// TIA Portal V21 export
TYPE "OBJ_Washing_Phase_V100_Type"
   STRUCT
      x_Start_Ok : Bool;   // 0.2 - Consenso Inizio Fase
      x_EN_Next_Step : Bool;   // 0.3 - Abilita Passo Successivo (al pastorizzatore)
      Free04 : Bool;
      x_Aux_Next_Step_After_Drain : Bool;   // 0.5 - Aux Passo Successivo Dopo Drenaggio
      x_Start_Step_Mngr : Bool;   // 0.6 - InizioGestionePassi
      x_Stop_Step_Mngr : Bool;   // 0.7 - FineGestionePassi
      x_AppFP_Start : Bool;   // 1.0 - AppoggioFrInizio
      x_Pulse_Start : Bool;   // 1.1 - FronteInizio
   END_STRUCT;
END_TYPE
